{attribute addProperty BoxType "EK1960-0000-0021"}
{attribute addProperty Id "FSOEAT %Q*FSOE_B358BD5C12015"}
{attribute addProperty CRC "3675236599"}
{attribute addProperty SizeInBites "120"}
{attribute addProperty SizeInBytes "15"}
TYPE FSoE_Outputs_DB0FA8F7 :
STRUCT
	{attribute addProperty Name "FSOE"}
	FSOE AT %Q* : FSOE_B358BD5C;
END_STRUCT
END_TYPE

(* stored: Version 1.2.0.0, ProductVersion 3.1.4024.9
   DUT FSoE_Outputs_DB0FA8F7: Id {8d1f88ed-8529-4cb6-860a-9e0012b16fb9} *)
